PROGRAM F_EndschalterBruecken
VAR
	
END_VAR

(* Baustein: FC2 Start, Stop, Betriebsarten *)
(* Netzwerk: 1 Endschalter brücken *)

(* Vorgehensweise: Eine bestimmte mögliche (Ausgangs-)Kombi wird meist etwas verzögert als Eingang 'dargeboten'... 
damit wird der entsprechende Eingang simuliert *)


(*
	U "M11.0_Bridge_E1.0" M11.0 -- Brücke E1.0 Drahthalter offen
	SPBN br10
	
	UN "A 1.7" A1.7 -- Y-10 Drahthalter+Führung zu
	L S5T#500MS
	SE "Bridge_E1.0" T110 -- Brücke E1.0 Drahthalter offen
	U "Bridge_E1.0" T110 -- Brücke E1.0 Drahthalter offen
	= "E1_0" E1.0 -- R Drahthalter offen
*)
IF RVL.sBrDrahthalterIstOffen THEN //Brücke E1.2 (neu) Drahthalter offen, VAT.M11.0
	GVL.tonDrahthaltOffen(IN := NOT IO.outY10DrahthaltFuehrungZU, PT := T#500MS);
	GVL.insecDrahthalterIstOffen := GVL.tonDrahthaltOffen.Q;
ELSE

	{IF defined (CRIMP_IO_TEST)}
		GVL.insecDrahthalterIstOffen := GVL.inTmpDrahthalterIstOffen;
	{ELSE}
		GVL.insecDrahthalterIstOffen := IO.inDrahthalterIstOffen;
	{END_IF}	
	
END_IF

(*	
br10:
	U "M11.1_Bridge_E1.1" M11.1 -- Brücke E1.1 Auslöseschalter
	SPBN br11
	U "A 0.0" A0.0 -- Tastleuchte Start
	O "M0_3_Tipp" M0.3 -- Einzel-Schritt
	U "M 80.0" M80.0 -- +F E0.0 Taste Start
	= "E1_1" E1.1 -- N Auslöseschalter
*)
IF RVL.sBrAusloeseSchalter THEN //Brücke E1.3 (neu) Auslöseschalter, war VAT.M11.1
	GVL.insecAusloeseSchalter := IO.outMldTasteStart OR VAT.bEinzelSchritt AND VAT.bFlkTasteStart;
ELSE
	{IF defined (CRIMP_IO_TEST)}
		GVL.insecAusloeseSchalter := GVL.inTmpAusloeseSchalter;
	{ELSE}
		GVL.insecAusloeseSchalter := IO.inAusloeseSchalter;
	{END_IF}
END_IF
(*
br11:
	U "M11.2_Bridge_E1.2" M11.2 -- Brücke E1.2 Abisolierer zu
	SPBN br12
	U "A 1.3" A1.3 -- Y-6 Abisolierer zu
	L S5T#300MS
	SE "Bridge_E1.2" T112 -- Brücke E1.2 Abisolierer zu
	U "Bridge_E1.2" T112 -- Brücke E1.2 Abisolierer zu
	= "E1_2" E1.2 -- N Abisolierer zu
*)
IF RVL.sBrAbisoliererIstZU THEN //Brücke E1.4 (neu) Auslöseschalter, war VAT.M11.2
	GVL.tonAbisoliererIstZU(IN := IO.outY6AbisoliererZU, PT := T#300MS); // war T112
	GVL.insecAbisoliererIstZU := GVL.tonAbisoliererIstZU.Q;
ELSE	
	{IF defined (CRIMP_IO_TEST)}
		GVL.insecAbisoliererIstZU := GVL.inTmpAbisoliererIstZU;
	{ELSE}
		GVL.insecAbisoliererIstZU := IO.inAbisoliererIstZU;
	{END_IF}
END_IF
(*
br12: U "M11.3_Bridge_E1.3" M11.3 -- Brücke E1.3 Abisolierer vorn
	SPBN br13
	UN "A 1.5" A1.5 -- Y-8 Abisolierer rück
	L S5T#300MS
	SE "Bridge_E1.3" T113 -- Brücke E1.3 Abisolierer vorn
	U "Bridge_E1.3" T113 -- Brücke E1.3 Abisolierer vorn
	= "E1_3" E1.3 -- R Abisolierer vorn
*)
IF RVL.sBrAbisoliererIstVORN THEN //Brücke E1.5 (neu) Abisolierer vorn, war VAT.M11.3
	GVL.tonAbisoliererIstVORN(IN := NOT IO.outY8AbisoliererRUECK, PT := T#300MS); // war T113
	GVL.insecAbisoliererIstVORN := GVL.tonAbisoliererIstVORN.Q;
ELSE
	{IF defined (CRIMP_IO_TEST)}
		GVL.insecAbisoliererIstVORN := GVL.inTmpAbisoliererIstVORN;
	{ELSE}	
		GVL.insecAbisoliererIstVORN := IO.inAbisoliererIstVORN;
	{END_IF}	
END_IF
(*
br13: U "M11.4_Bridge_E1.4" M11.4 -- Brücke E1.4 Abisolierer rück (abisoliert)
	SPBN br14
	U "A 1.5" A1.5 -- Y-8 Abisolierer rück
	L S5T#400MS
	SE "Bridge_E1.4" T114 -- Brücke E1.4 Abisolierer rück (abisoliert)
	U "Bridge_E1.4" T114 -- Brücke E1.4 Abisolierer rück (abisoliert)
	= "E1_4" E1.4 -- R Abisolierer rück (abisoliert)
*)
IF RVL.sBrAbisoliererIstRUECK THEN //Brücke E1.6 (neu) Abisolierer rück (abisoliert), war VAT.M11.4
	GVL.tonAbisoliererIstRUECK(IN := IO.outY8AbisoliererRUECK, PT := T#400MS); // war T114
	GVL.insecAbisoliererIstRUECK := GVL.tonAbisoliererIstRUECK.Q;
ELSE
	{IF defined (CRIMP_IO_TEST)}
		GVL.insecAbisoliererIstRUECK := GVL.inTmpAbisoliererIstRUECK;
	{ELSE}	
		GVL.insecAbisoliererIstRUECK := IO.inAbisoliererIstRUECK;
	{END_IF}	
END_IF
(*
br14: U "M11.5_Bridge_E1.5" M11.5 -- Brücke E1.5 Abisolierer links (aus Arbeitsraum)
	SPBN br15
	U "A 1.2" A1.2 -- Y-5 Abisolierer nach links+Abdeckung zu
	L S5T#500MS
	SE "Bridge_E1.5" T115 -- Brücke E1.5 Abisolierer links (aus Arbeitsraum)
	U "Bridge_E1.5" T115 -- Brücke E1.5 Abisolierer links (aus Arbeitsraum)
	= "E1_5" E1.5 -- R Abisolierer links (aus Arbeitsraum)
*)
IF RVL.sBrAbisoliererIstLINKS THEN //Brücke E1.7 (neu) Abisolierer links (aus Arbeitsraum), war VAT.M11.5
	GVL.tonAbisoliererIstLINKS(IN := IO.outY5AbisolierNachLINKS, PT := T#500MS); // war T115
	GVL.insecAbisoliererIstLINKS := GVL.tonAbisoliererIstLINKS.Q;
ELSE
	{IF defined (CRIMP_IO_TEST)}
		GVL.insecAbisoliererIstLINKS := GVL.inTmpAbisoliererIstLINKS;
	{ELSE}	
		GVL.insecAbisoliererIstLINKS := IO.inAbisoliererIstLINKS;
	{END_IF}	
END_IF
(*
br15: U "M11.6_Bridge_E1.6" M11.6 -- Brücke E1.6 Crimpzange zu
	SPBN br16
	U "A 1.6" A1.6 -- Y-9 Crimpen zu
	L S5T#600MS
	SE "Bridge_E1.6" T116 -- Brücke E1.6 Crimpzange zu
	U "Bridge_E1.6" T116 -- Brücke E1.6 Crimpzange zu
	= "E1_6" E1.6 -- N Crimpzange zu
*)
IF RVL.sBrCrimpZangeIstZU THEN //Brücke E1.8 (neu) Crimpzange zu, war VAT.M11.6
	GVL.tonCrimpZangeIstZU(IN := IO.outY9CrimperZU, PT := T#600MS); // war T116
	GVL.insecCrimpZangeIstZU := GVL.tonCrimpZangeIstZU.Q;
ELSE	
	{IF defined (CRIMP_IO_TEST)}
		GVL.insecCrimpZangeIstZU := GVL.inTmpCrimpZangeIstZU;
	{ELSE}	
		GVL.insecCrimpZangeIstZU := IO.inCrimpZangeIstZU;
	{END_IF}
END_IF
(*
br16: U "M11.7_Bridge_E1.7" M11.7 -- Brücke E1.7 Crimpzange offen
	SPBN br17
	UN "A 1.6" A1.6 -- Y-9 Crimpen zu
	L S5T#400MS
	SE "Bridge_E1.7" T117 -- Brücke E1.7 Crimpzange offen
	U "Bridge_E1.7" T117 -- Brücke E1.7 Crimpzange offen
	= "E1_7" E1.7 -- R Crimpzange offen
*)
IF RVL.sBrCrimpZangeIstOFFEN THEN //Brücke E1.9 (neu) Crimpzange offen, war VAT.M11.7
	GVL.tonCrimpZangeIstOFFEN(IN := NOT IO.outY9CrimperZU, PT := T#400MS); // war T117
	GVL.insecCrimpZangeIstOFFEN := GVL.tonCrimpZangeIstOFFEN.Q;
ELSE
	{IF defined (CRIMP_IO_TEST)}
		GVL.insecCrimpZangeIstOFFEN := GVL.inTmpCrimpZangeIstOFFEN;
	{ELSE}	
		GVL.insecCrimpZangeIstOFFEN := IO.inCrimpZangeIstOFFEN;
	{END_IF}	
END_IF
(*
br17: U "M12.0_Bridge_E2.0" M12.0 -- Brücke E2.0 Kontakt gefallen
	SPBN br20
	U "M 21.7" M21.7 -- Kontakt-Anforderung
	L S5T#500MS
	SE "Bridge_E2.0" T120 -- Brücke E2.0 Kontakt gefallen
	U "Bridge_E2.0" T120 -- Brücke E2.0 Kontakt gefallen
	= "E2_0" E2.0 -- L Kontakt gefallen
*)
IF RVL.sBrKontaktIstGefallen THEN //Brücke E1.10 (neu) Kontakt gefallen, war VAT.M12.0
	GVL.tonBrKontaktIstGefallen(IN := VAT.bKontaktAnforderung, PT := T#500MS); // war T120 -> M21.7
	GVL.insecKontaktIstGefallen := GVL.tonBrKontaktIstGefallen.Q;
ELSE	
	{IF defined (CRIMP_IO_TEST)}
		GVL.insecKontaktIstGefallen := GVL.inTmpKontaktIstGefallen;
	{ELSE}	
		GVL.insecKontaktIstGefallen := IO.inKontaktIstGefallen;
	{END_IF}
END_IF
(*
br20: U "M12.1_Bridge_E2.1" M12.1 -- Brücke E2.1 Crimpeinheit vorn
	SPBN br21
	U "A 1.1" A1.1 -- Y-4 Crimpeinheit vor
	L S5T#300MS
	SE "Bridge_E2.1" T121 -- Brücke E2.1 Crimpeinheit vorn
	U "Bridge_E2.1" T121 -- Brücke E2.1 Crimpeinheit vorn
	= "E2_1" E2.1 -- R Crimpeinheit vorn
*)
IF RVL.sBrCrimpEinheitIstVORN THEN //Brücke E1.11 (neu) Crimpeinheit vorn, war VAT.M12.1
	GVL.tonCrimpEinheitIstVORN(IN := IO.outY4CrimpEinheitVOR, PT := T#300MS); // war T121
	GVL.insecCrimpEinheitIstVORN := GVL.tonCrimpEinheitIstVORN.Q;
ELSE	
	{IF defined (CRIMP_IO_TEST)}
		GVL.insecCrimpEinheitIstVORN := GVL.inTmpCrimpEinheitIstVORN;
	{ELSE}	
		GVL.insecCrimpEinheitIstVORN := IO.inCrimpEinheitIstVORN;
	{END_IF}	
END_IF
(*
br21: U "M12.2_Bridge_E2.2" M12.2 -- Brücke E2.2 Kontakt-Schieben vorn
	SPBN br22
	U "A 1.0" A1.0 -- Y-3 Kontakt-Schieben
	L S5T#400MS
	SE "Bridge_E2.2" T122 -- Brücke E2.2 Kontakt-Schieben vorn
	U "Bridge_E2.2" T122 -- Brücke E2.2 Kontakt-Schieben vorn
	= "E2_2" E2.2 -- R Kontakt-Schieben vorn
*)
IF RVL.sBrKontaktSchiebenVORN THEN //Brücke E1.14 (neu) Kontakt-Schieben vorn, war VAT.M12.2
	GVL.tonKontaktSchiebenVORN(IN := IO.outY3KontaktSchieben, PT := T#400MS); // war T122
	GVL.insecKontaktSchiebenVORN := GVL.tonKontaktSchiebenVORN.Q;
ELSE	
	{IF defined (CRIMP_IO_TEST)}
		GVL.insecKontaktSchiebenVORN := GVL.inTmpKontaktSchiebenVORN;
	{ELSE}
		GVL.insecKontaktSchiebenVORN := IO.inKontaktSchiebenVORN;
	{END_IF}
END_IF
(*
br22: U "M12.3_Bridge_E2.3" M12.3 -- Brücke E2.3 Ausstoßen vorn
	SPBN br23
	U "A 0.6" A0.6 -- Y-1 Ausstoßen
	L S5T#300MS
	SE "Bridge_E2.3" T123 -- Brücke E2.3 Ausstoßen vorn
	U "Bridge_E2.3" T123 -- Brücke E2.3 Ausstoßen vorn
	= "E2_3" E2.3 -- R Ausstoßen vorn
*)
IF RVL.sBrAusstossenVORN THEN //Brücke E1.13 (neu) Ausstoßen vorn, war VAT.M12.3
	GVL.tonAusstossenVORN(IN := IO.outY1Ausstossen, PT := T#300MS); // war T123
	GVL.insecAusstossenVORN := GVL.tonAusstossenVORN.Q;
ELSE
	{IF defined (CRIMP_IO_TEST)}
		GVL.insecAusstossenVORN := GVL.inTmpAusstossenVORN;
	{ELSE}	
		GVL.insecAusstossenVORN := IO.inAusstossenVORN;
	{END_IF}
END_IF
(*
br23: U "M12.4_Bridge_E2.4" M12.4 -- Brücke E2.4 Crimpeinheit rück
	SPBN br24
	UN "A 1.1" A1.1 -- Y-4 Crimpeinheit vor
	L S5T#400MS
	SE "Bridge_E2.4" T124 -- Brücke E2.4 Crimpeinheit rück
	U "Bridge_E2.4" T124 -- Brücke E2.4 Crimpeinheit rück
	= "E2_4" E2.4 -- R Crimpeinheit rück
*)
IF RVL.sBrAusstossenVORN THEN //Brücke E1.12 (neu) Crimpeinheit rück, war VAT.M12.4
	GVL.tonCrimpEinheitIstRUECK(IN := IO.outY4CrimpEinheitVOR, PT := T#300MS); // war T124
	GVL.insecCrimpEinheitIstRUECK := GVL.tonCrimpEinheitIstRUECK.Q;
ELSE
	{IF defined (CRIMP_IO_TEST)}
		GVL.insecCrimpEinheitIstRUECK := GVL.inTmpCrimpEinheitIstRUECK;
	{ELSE}
		GVL.insecCrimpEinheitIstRUECK := IO.inCrimpEinheitIstRUECK;
	{END_IF}	
END_IF
(*
br24: U "M12.5_Bridge_E2.5" M12.5 -- Brücke E2.5 Magazin gefüllt
	SPBN br25
	U "E2_5" E2.5 -- N Magazin gefüllt
	= "E2_5" E2.5 -- N Magazin gefüllt
*)
IF RVL.sBrMagazinGEFUELLT THEN // //Brücke E1.15 (neu) Magazin gefüllt, war VAT.M12.5
	GVl.insecMagazinGEFUELLT := IO.inMagazinGEFUELLT; //???
ELSE	
	{IF defined (CRIMP_IO_TEST)}
		GVL.insecMagazinGEFUELLT := GVL.inTmpMagazinGEFUELLT;
	{ELSE}
		GVl.insecMagazinGEFUELLT := IO.inMagazinGEFUELLT;
	{END_IF}	
END_IF
(*
br25: BLD 130
*)

END_PROGRAM

(* stored: Version 1.1.0.1, ProductVersion 3.1.4024.3
   POU F_EndschalterBruecken: Id {b93c4c15-18fb-49a5-bc3a-e39cc8e09da8}, SpecialFunc None *)
